// String formatting helper namespace.
PROGRAM Strf

// Formats with one Tc2_Utilities argument.
METHOD Fmt : Str
VAR_INPUT
	sFormat			: Str; // Format string.
	tcArg			: Tc2_Utilities.T_Arg; // Format argument.
END_VAR
VAR
	_fmt			: Tc2_Utilities.FB_FormatString;
END_VAR
_fmt(sFormat := sFormat, arg1 := tcArg, sOut => Fmt);
END_METHOD

// Pads text; returns padded value.
METHOD Padding : Str
VAR_INPUT
    sValue       : Str;  // Text to pad.
    nLeftPadding : USINT := 0; // Minimum left-padded width.
    nRightPadding: USINT := 0; // Minimum right-padded width.
    sFillChar    : Ch := ' ';  // Fill character.
END_VAR
VAR
	_nLen		: INT := Tc2_Standard.LEN(sValue);
	_nLeftMiss	: INT;
	_nRightMiss	: INT;	

	i			: INT;
END_VAR
_nLeftMiss := nLeftPadding - _nLen;
_nRightMiss := nRightPadding - _nLen;

IF _nLeftMiss > 0 THEN
	FOR i := 1 TO _nleftMiss DO
		sValue := Tc2_Standard.CONCAT(sFillChar, sValue);
	END_FOR	
END_IF

IF _nRightMiss > 0 THEN
	FOR i := 1 TO _nRightMiss DO
		sValue := Tc2_Standard.CONCAT(sFillChar, sValue);
	END_FOR	
END_IF

Padding := sValue;
END_METHOD

// Formats TIME; returns empty string on invalid unit range.
METHOD SimpleTime : Str
VAR_INPUT
    tValue   : TIME;  // Time to format.
    sMinUnit : Str := 'MS'; // Minimum unit: MS, S, M, H, or D.
    sMaxUnit : Str := 'S';  // Maximum unit: MS, S, M, H, or D.
END_VAR
VAR
	_nMinUnit	: USINT;
	_nMaxUnit	: USINT;
	_sValues	: ARRAY[1..5] OF Strb;
	_nValues	: ARRAY[1..5] OF UINT;
	_sUnits   	: ARRAY[1..5] OF STRING := ['MS', 'S', 'M', 'H', 'D'];
	_stTime		: Tc2_Utilities.OTSTRUCT;
	_i			: USINT;
	_strb		: Strb;
END_VAR
FOR _i := 1 TO 5 DO
	IF _sUnits[_i] = sMinUnit THEN
		_nMinUnit := _i;
	END_IF
	IF _sUnits[_i] = sMaxUnit THEN
		_nMaxUnit := _i;
	END_IF
END_FOR

IF _nMaxUnit = 0 THEN
	RETURN;
END_IF

IF _nMinUnit = 0 THEN
	RETURN;
END_IF

IF _nMinUnit > _nMaxUnit THEN
	RETURN;
END_IF

_stTime := Tc2_Utilities.TIME_TO_OTSTRUCT(tValue);
_stTime.wDay := _stTime.wWeek * 7 + _stTime.wDay;

_nValues[1] := WORD_TO_UINT(_stTime.wMilliseconds);
_nValues[2] := WORD_TO_UINT(_stTime.wSecond);
_nValues[3] := WORD_TO_UINT(_stTime.wMinute);
_nValues[4] := WORD_TO_UINT(_stTime.wHour);
_nValues[5] := WORD_TO_UINT(_stTime.wDay);

_sValues[1].Set(Strf.Padding(UINT_TO_STRING(_nValues[1]), 3, 0, '0')).Append('ms');
_sValues[2].Set(Strf.Padding(UINT_TO_STRING(_nValues[2]), 2, 0, '0')).Append('s');
_sValues[3].Set(Strf.Padding(UINT_TO_STRING(_nValues[3]), 2, 0, '0')).Append('m');
_sValues[4].Set(Strf.Padding(UINT_TO_STRING(_nValues[4]), 2, 0, '0')).Append('h');
_sValues[5].Set(Strf.Padding(UINT_TO_STRING(_nValues[5]), 3, 0, '0')).Append('d');

IF _nMaxUnit < 5 THEN
    FOR _i := 5 TO _nMaxUnit + 1 BY -1 DO
        IF _nValues[_i] <> 0 THEN
            _strb.Append(_sValues[_i].Get()).Append(' ');
        END_IF
    END_FOR
END_IF

FOR _i := _nMaxUnit TO _nMinUnit BY -1 DO
    _strb.Append(_sValues[_i].Get()).Append(' ');
END_FOR

SimpleTime := _strb.Get();
END_METHOD

END_PROGRAM

(* stored: Version 1.1.0.1
   POU Strf: Id {1997d8f8-a3a3-412e-a9d9-e47c6d4dafb7}, SpecialFunc None
   Method Fmt: Id {2e4699c7-d42c-40f8-a916-1ba18101d5a2}
   Method Padding: Id {7d05623e-05a9-49ee-b8ca-0efb8661641b}
   Method SimpleTime: Id {2c25983c-5b99-43fa-a5a9-faa93b5102ab} *)
